FUNCTION_BLOCK Q_NumericValue (* Command change numeric value ( Part 6 - F.22 ) *)
  (* Standard: ISO 11783-6; Description: This command is used to change the value of an object. It applies only to objects that have a numeric value attribute. Return values iso_s16 - E_NO_ERR - OK - E_OVERFLOW - buffer overflow - E_NOACT - Command not possible in current state - E_NO_INSTANCE - No VT client available *)
  (* Version 1.0, 2022-07-08, franz *)
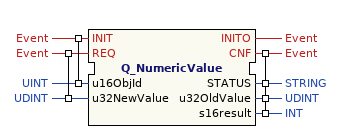
  EVENT_INPUT
    INIT WITH u16ObjId; (* Service Initialization *)
    REQ WITH u32NewValue; (* Service Request *)
  END_EVENT
  EVENT_OUTPUT
    INITO; (* Initialization Confirm *)
    CNF WITH STATUS, u32OldValue, s16result; (* Confirmation of Requested Service *)
  END_EVENT
  VAR_INPUT
    u16ObjId : UINT; (* Object ID *)
    u32NewValue : UDINT; (* New value of ID *)
  END_VAR
  VAR_OUTPUT
    STATUS : STRING; (* Service Status *)
    u32OldValue : UDINT; (* Old value of ID *)
    s16result : INT; (* retval see description *)
  END_VAR
END_FUNCTION_BLOCK
